// TIA Portal V20 export
FUNCTION_BLOCK "PartData"   // FB50063, LAD
// stored: MemoryReserve 100, Namespace Unit1.Em7, SetENOAutomatically false
   VAR
      statPulse { ExternalAccessible := 'False'; ExternalVisible := 'False'; ExternalWritable := 'False'} : Array[0..99] of Bool;
   END_VAR
   VAR_TEMP
      tempRetVal : Int;
   END_VAR
   VAR_TEMP   // added for the SCL form of the ladder/FBD networks
      _w1 : Bool;
      _w2 : Bool;
      _w3 : Bool;
      _w4 : Bool;
   END_VAR
BEGIN

REGION Network 1: Stack Table → Sepa Gripper
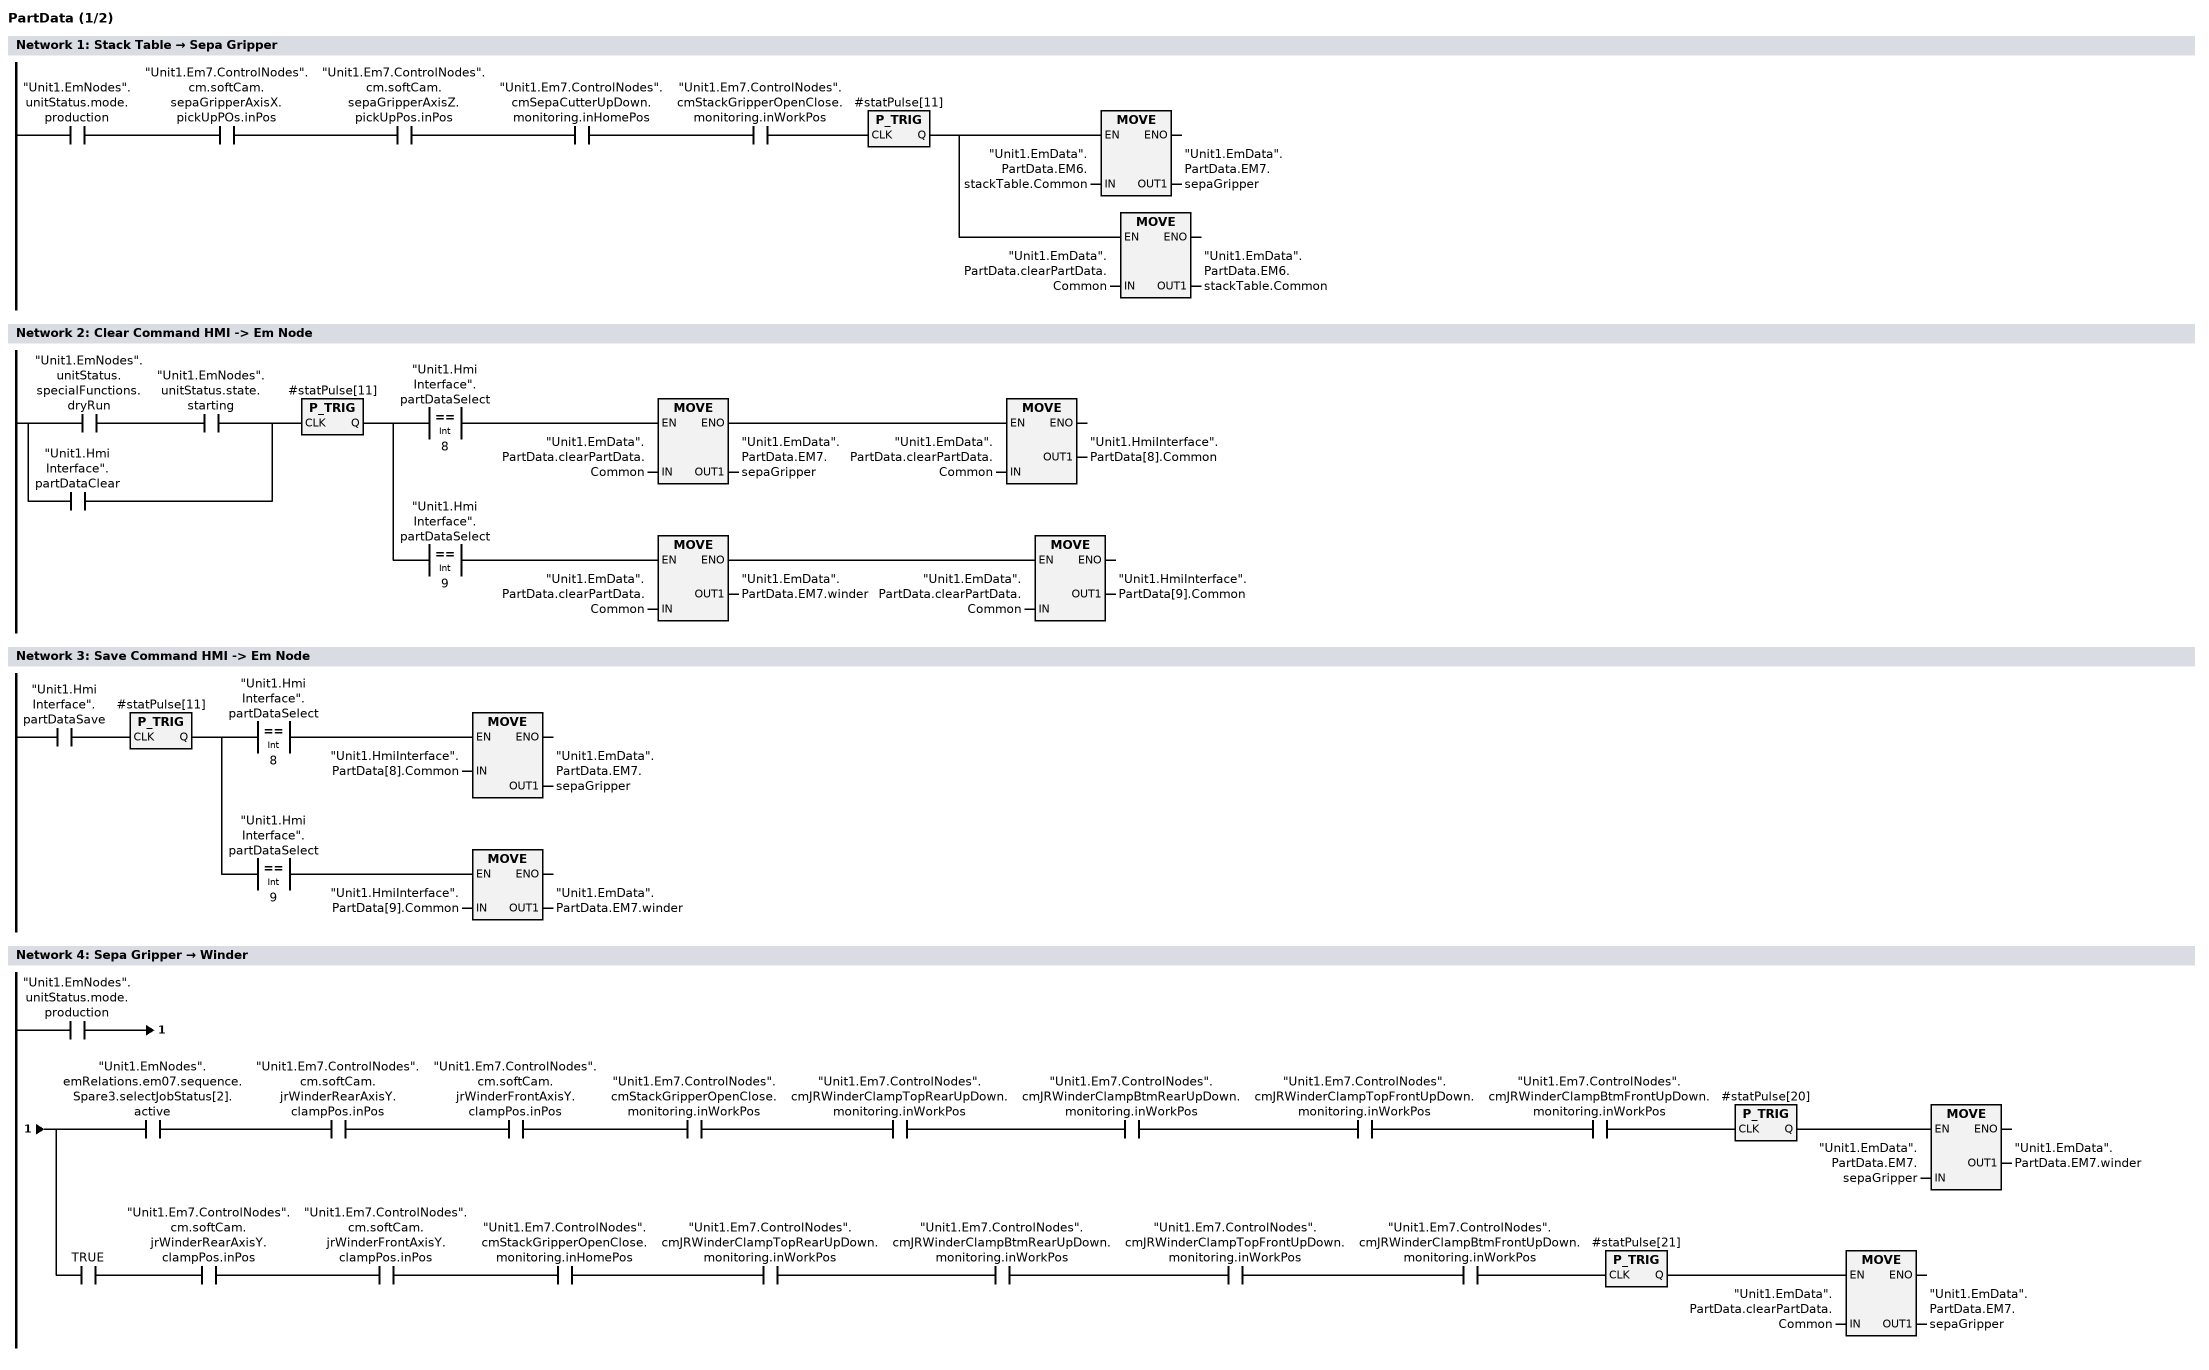
   RUNG wire#powerrail
      Contact( "Unit1.EmNodes".unitStatus.mode.production )
      Contact( "Unit1.Em7.ControlNodes".cm.softCam.sepaGripperAxisX.pickUpPOs.inPos )
      Contact( "Unit1.Em7.ControlNodes".cm.softCam.sepaGripperAxisZ.pickUpPos.inPos )
      Contact( "Unit1.Em7.ControlNodes".cmSepaCutterUpDown.monitoring.inHomePos )
      Contact( "Unit1.Em7.ControlNodes".cmStackGripperOpenClose.monitoring.inWorkPos )
      P_Trig( #statPulse[11] )
      wire#w1
      Move(in := "Unit1.EmData".PartData.EM6.stackTable.Common, out1 => "Unit1.EmData".PartData.EM7.sepaGripper)
   END_RUNG
   RUNG wire#w1
      Move(in := "Unit1.EmData".PartData.clearPartData.Common, out1 => "Unit1.EmData".PartData.EM6.stackTable.Common)
   END_RUNG
   // the same network as SCL:
   #_w1 := "Unit1.EmNodes".unitStatus.mode.production AND "Unit1.Em7.ControlNodes".cm.softCam.sepaGripperAxisX.pickUpPOs.inPos AND "Unit1.Em7.ControlNodes".cm.softCam.sepaGripperAxisZ.pickUpPos.inPos AND "Unit1.Em7.ControlNodes".cmSepaCutterUpDown.monitoring.inHomePos AND "Unit1.Em7.ControlNodes".cmStackGripperOpenClose.monitoring.inWorkPos;
   #_w2 := #_w1 AND NOT #statPulse[11];   // rising edge
   #statPulse[11] := #_w1;
   IF #_w2 THEN
       "Unit1.EmData".PartData.EM7.sepaGripper := "Unit1.EmData".PartData.EM6.stackTable.Common;
       "Unit1.EmData".PartData.EM6.stackTable.Common := "Unit1.EmData".PartData.clearPartData.Common;
   END_IF;
END_REGION

REGION Network 2: Clear Command HMI -> Em Node
   RUNG wire#powerrail
      Contact( "Unit1.EmNodes".unitStatus.specialFunctions.dryRun )
      Contact( "Unit1.EmNodes".unitStatus.state.starting )
      wire#w1
      P_Trig( #statPulse[11] )
      wire#w2
      { S7_Templates := "SrcType := Int" } EQ_Contact(in1 := "Unit1.HmiInterface".partDataSelect, in2 := 8)
      Move(in := "Unit1.EmData".PartData.clearPartData.Common, out1 => "Unit1.EmData".PartData.EM7.sepaGripper)
      Move(in := "Unit1.EmData".PartData.clearPartData.Common, out1 => "Unit1.HmiInterface".PartData[8].Common)
   END_RUNG
   RUNG wire#powerrail
      Contact( "Unit1.HmiInterface".partDataClear )
   END_RUNG wire#w1
   RUNG wire#w2
      { S7_Templates := "SrcType := Int" } EQ_Contact(in1 := "Unit1.HmiInterface".partDataSelect, in2 := 9)
      Move(in := "Unit1.EmData".PartData.clearPartData.Common, out1 => "Unit1.EmData".PartData.EM7.winder)
      Move(in := "Unit1.EmData".PartData.clearPartData.Common, out1 => "Unit1.HmiInterface".PartData[9].Common)
   END_RUNG
   // the same network as SCL:
   #_w1 := ("Unit1.EmNodes".unitStatus.specialFunctions.dryRun AND "Unit1.EmNodes".unitStatus.state.starting) OR "Unit1.HmiInterface".partDataClear;
   #_w2 := #_w1 AND NOT #statPulse[11];   // rising edge
   #statPulse[11] := #_w1;
   IF #_w2 AND ("Unit1.HmiInterface".partDataSelect = 8) THEN
       "Unit1.EmData".PartData.EM7.sepaGripper := "Unit1.EmData".PartData.clearPartData.Common;
       "Unit1.HmiInterface".PartData[8].Common := "Unit1.EmData".PartData.clearPartData.Common;
   END_IF;
   IF #_w2 AND ("Unit1.HmiInterface".partDataSelect = 9) THEN
       "Unit1.EmData".PartData.EM7.winder := "Unit1.EmData".PartData.clearPartData.Common;
       "Unit1.HmiInterface".PartData[9].Common := "Unit1.EmData".PartData.clearPartData.Common;
   END_IF;
END_REGION

REGION Network 3: Save Command HMI -> Em Node
   RUNG wire#powerrail
      Contact( "Unit1.HmiInterface".partDataSave )
      P_Trig( #statPulse[11] )
      wire#w1
      { S7_Templates := "SrcType := Int" } EQ_Contact(in1 := "Unit1.HmiInterface".partDataSelect, in2 := 8)
      Move(in := "Unit1.HmiInterface".PartData[8].Common, out1 => "Unit1.EmData".PartData.EM7.sepaGripper)
   END_RUNG
   RUNG wire#w1
      { S7_Templates := "SrcType := Int" } EQ_Contact(in1 := "Unit1.HmiInterface".partDataSelect, in2 := 9)
      Move(in := "Unit1.HmiInterface".PartData[9].Common, out1 => "Unit1.EmData".PartData.EM7.winder)
   END_RUNG
   // the same network as SCL:
   #_w1 := "Unit1.HmiInterface".partDataSave AND NOT #statPulse[11];   // rising edge
   #statPulse[11] := "Unit1.HmiInterface".partDataSave;
   IF #_w1 AND ("Unit1.HmiInterface".partDataSelect = 8) THEN
       "Unit1.EmData".PartData.EM7.sepaGripper := "Unit1.HmiInterface".PartData[8].Common;
   END_IF;
   IF #_w1 AND ("Unit1.HmiInterface".partDataSelect = 9) THEN
       "Unit1.EmData".PartData.EM7.winder := "Unit1.HmiInterface".PartData[9].Common;
   END_IF;
END_REGION

REGION Network 4: Sepa Gripper → Winder
   RUNG wire#powerrail
      Contact( "Unit1.EmNodes".unitStatus.mode.production )
      wire#w1
      Contact( "Unit1.EmNodes".emRelations.em07.sequence.Spare3.selectJobStatus[2].active )
      Contact( "Unit1.Em7.ControlNodes".cm.softCam.jrWinderRearAxisY.clampPos.inPos )
      Contact( "Unit1.Em7.ControlNodes".cm.softCam.jrWinderFrontAxisY.clampPos.inPos )
      Contact( "Unit1.Em7.ControlNodes".cmStackGripperOpenClose.monitoring.inWorkPos )
      Contact( "Unit1.Em7.ControlNodes".cmJRWinderClampTopRearUpDown.monitoring.inWorkPos )
      Contact( "Unit1.Em7.ControlNodes".cmJRWinderClampBtmRearUpDown.monitoring.inWorkPos )
      Contact( "Unit1.Em7.ControlNodes".cmJRWinderClampTopFrontUpDown.monitoring.inWorkPos )
      Contact( "Unit1.Em7.ControlNodes".cmJRWinderClampBtmFrontUpDown.monitoring.inWorkPos )
      P_Trig( #statPulse[20] )
      Move(in := "Unit1.EmData".PartData.EM7.sepaGripper, out1 => "Unit1.EmData".PartData.EM7.winder)
   END_RUNG
   RUNG wire#w1
      Contact( TRUE )
      Contact( "Unit1.Em7.ControlNodes".cm.softCam.jrWinderRearAxisY.clampPos.inPos )
      Contact( "Unit1.Em7.ControlNodes".cm.softCam.jrWinderFrontAxisY.clampPos.inPos )
      Contact( "Unit1.Em7.ControlNodes".cmStackGripperOpenClose.monitoring.inHomePos )
      Contact( "Unit1.Em7.ControlNodes".cmJRWinderClampTopRearUpDown.monitoring.inWorkPos )
      Contact( "Unit1.Em7.ControlNodes".cmJRWinderClampBtmRearUpDown.monitoring.inWorkPos )
      Contact( "Unit1.Em7.ControlNodes".cmJRWinderClampTopFrontUpDown.monitoring.inWorkPos )
      Contact( "Unit1.Em7.ControlNodes".cmJRWinderClampBtmFrontUpDown.monitoring.inWorkPos )
      P_Trig( #statPulse[21] )
      Move(in := "Unit1.EmData".PartData.clearPartData.Common, out1 => "Unit1.EmData".PartData.EM7.sepaGripper)
   END_RUNG
   // the same network as SCL:
   #_w1 := "Unit1.EmNodes".unitStatus.mode.production AND "Unit1.EmNodes".emRelations.em07.sequence.Spare3.selectJobStatus[2].active AND "Unit1.Em7.ControlNodes".cm.softCam.jrWinderRearAxisY.clampPos.inPos AND "Unit1.Em7.ControlNodes".cm.softCam.jrWinderFrontAxisY.clampPos.inPos AND "Unit1.Em7.ControlNodes".cmStackGripperOpenClose.monitoring.inWorkPos AND "Unit1.Em7.ControlNodes".cmJRWinderClampTopRearUpDown.monitoring.inWorkPos AND "Unit1.Em7.ControlNodes".cmJRWinderClampBtmRearUpDown.monitoring.inWorkPos AND "Unit1.Em7.ControlNodes".cmJRWinderClampTopFrontUpDown.monitoring.inWorkPos AND "Unit1.Em7.ControlNodes".cmJRWinderClampBtmFrontUpDown.monitoring.inWorkPos;
   #_w2 := #_w1 AND NOT #statPulse[20];   // rising edge
   #statPulse[20] := #_w1;
   IF #_w2 THEN "Unit1.EmData".PartData.EM7.winder := "Unit1.EmData".PartData.EM7.sepaGripper; END_IF;
   #_w3 := "Unit1.EmNodes".unitStatus.mode.production AND TRUE AND "Unit1.Em7.ControlNodes".cm.softCam.jrWinderRearAxisY.clampPos.inPos AND "Unit1.Em7.ControlNodes".cm.softCam.jrWinderFrontAxisY.clampPos.inPos AND "Unit1.Em7.ControlNodes".cmStackGripperOpenClose.monitoring.inHomePos AND "Unit1.Em7.ControlNodes".cmJRWinderClampTopRearUpDown.monitoring.inWorkPos AND "Unit1.Em7.ControlNodes".cmJRWinderClampBtmRearUpDown.monitoring.inWorkPos AND "Unit1.Em7.ControlNodes".cmJRWinderClampTopFrontUpDown.monitoring.inWorkPos AND "Unit1.Em7.ControlNodes".cmJRWinderClampBtmFrontUpDown.monitoring.inWorkPos;
   #_w4 := #_w3 AND NOT #statPulse[21];   // rising edge
   #statPulse[21] := #_w3;
   IF #_w4 THEN
       "Unit1.EmData".PartData.EM7.sepaGripper := "Unit1.EmData".PartData.clearPartData.Common;
   END_IF;
END_REGION

REGION Network 5: Winder → Sepa Gripper
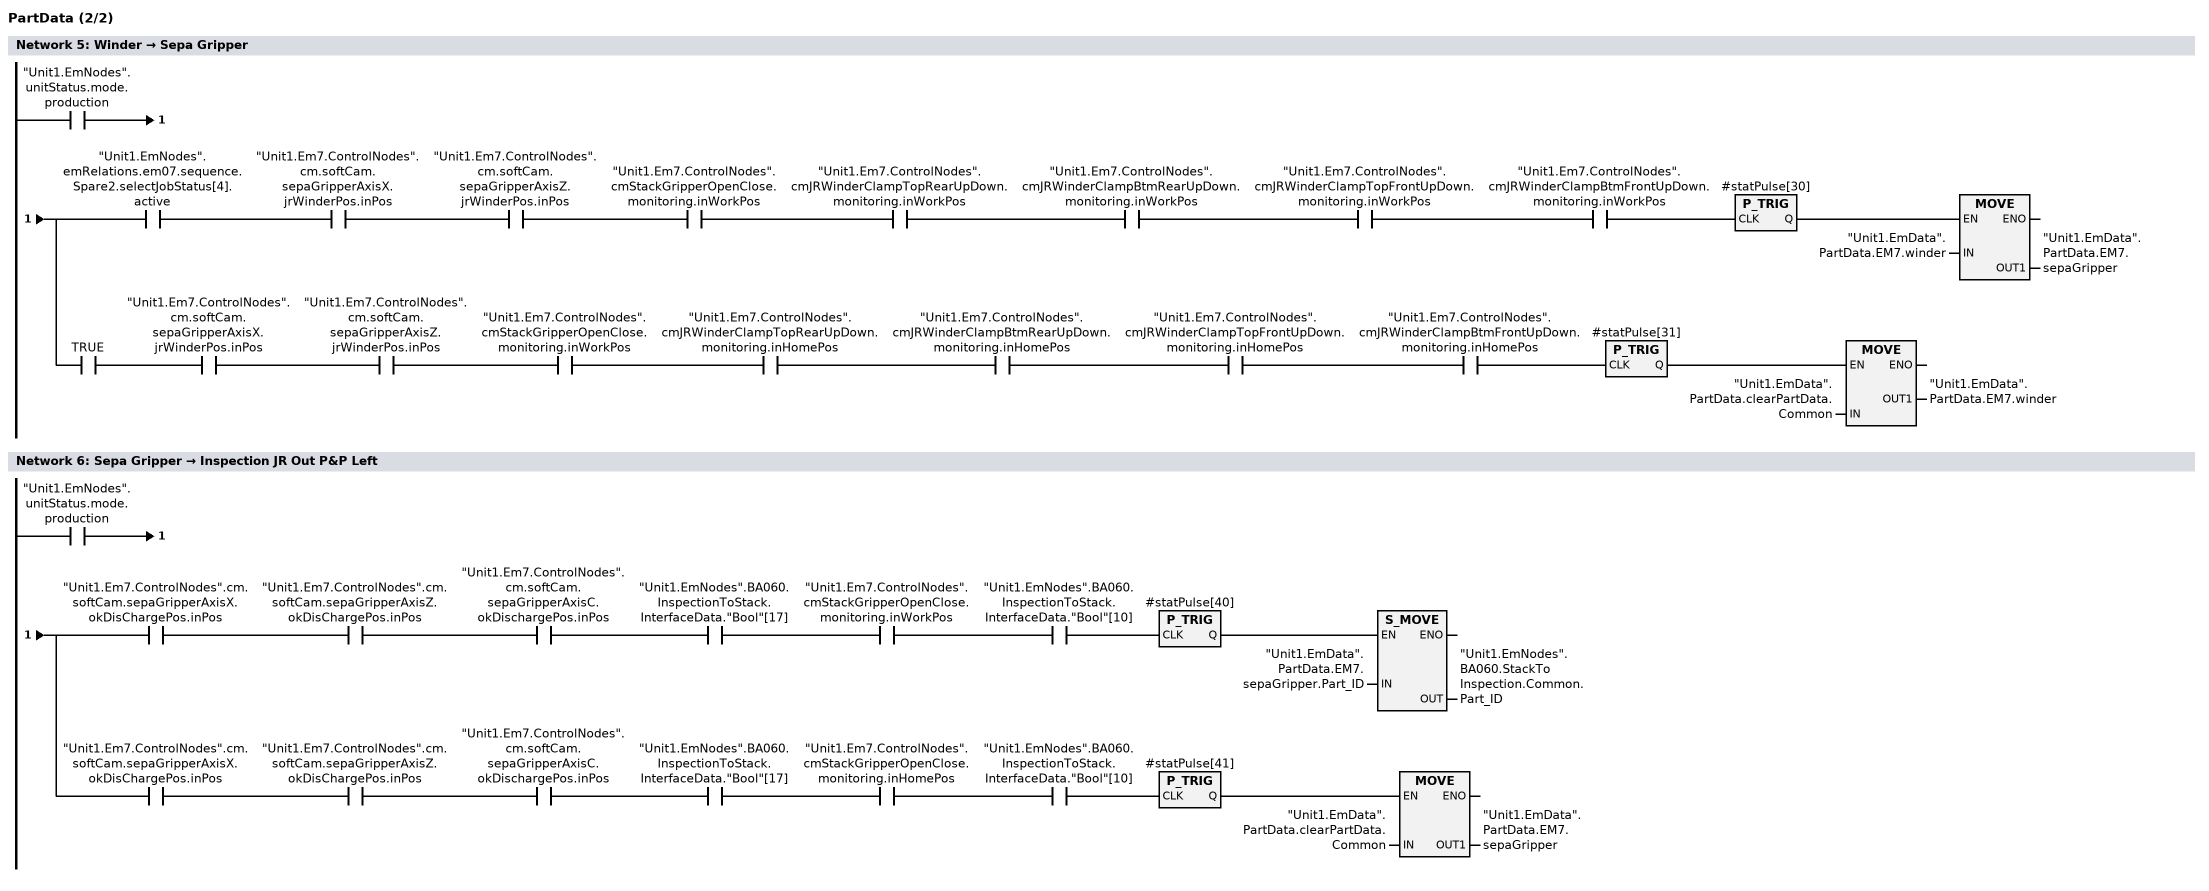
   RUNG wire#powerrail
      Contact( "Unit1.EmNodes".unitStatus.mode.production )
      wire#w1
      Contact( "Unit1.EmNodes".emRelations.em07.sequence.Spare2.selectJobStatus[4].active )
      Contact( "Unit1.Em7.ControlNodes".cm.softCam.sepaGripperAxisX.jrWinderPos.inPos )
      Contact( "Unit1.Em7.ControlNodes".cm.softCam.sepaGripperAxisZ.jrWinderPos.inPos )
      Contact( "Unit1.Em7.ControlNodes".cmStackGripperOpenClose.monitoring.inWorkPos )
      Contact( "Unit1.Em7.ControlNodes".cmJRWinderClampTopRearUpDown.monitoring.inWorkPos )
      Contact( "Unit1.Em7.ControlNodes".cmJRWinderClampBtmRearUpDown.monitoring.inWorkPos )
      Contact( "Unit1.Em7.ControlNodes".cmJRWinderClampTopFrontUpDown.monitoring.inWorkPos )
      Contact( "Unit1.Em7.ControlNodes".cmJRWinderClampBtmFrontUpDown.monitoring.inWorkPos )
      P_Trig( #statPulse[30] )
      Move(in := "Unit1.EmData".PartData.EM7.winder, out1 => "Unit1.EmData".PartData.EM7.sepaGripper)
   END_RUNG
   RUNG wire#w1
      Contact( TRUE )
      Contact( "Unit1.Em7.ControlNodes".cm.softCam.sepaGripperAxisX.jrWinderPos.inPos )
      Contact( "Unit1.Em7.ControlNodes".cm.softCam.sepaGripperAxisZ.jrWinderPos.inPos )
      Contact( "Unit1.Em7.ControlNodes".cmStackGripperOpenClose.monitoring.inWorkPos )
      Contact( "Unit1.Em7.ControlNodes".cmJRWinderClampTopRearUpDown.monitoring.inHomePos )
      Contact( "Unit1.Em7.ControlNodes".cmJRWinderClampBtmRearUpDown.monitoring.inHomePos )
      Contact( "Unit1.Em7.ControlNodes".cmJRWinderClampTopFrontUpDown.monitoring.inHomePos )
      Contact( "Unit1.Em7.ControlNodes".cmJRWinderClampBtmFrontUpDown.monitoring.inHomePos )
      P_Trig( #statPulse[31] )
      Move(in := "Unit1.EmData".PartData.clearPartData.Common, out1 => "Unit1.EmData".PartData.EM7.winder)
   END_RUNG
   // the same network as SCL:
   #_w1 := "Unit1.EmNodes".unitStatus.mode.production AND "Unit1.EmNodes".emRelations.em07.sequence.Spare2.selectJobStatus[4].active AND "Unit1.Em7.ControlNodes".cm.softCam.sepaGripperAxisX.jrWinderPos.inPos AND "Unit1.Em7.ControlNodes".cm.softCam.sepaGripperAxisZ.jrWinderPos.inPos AND "Unit1.Em7.ControlNodes".cmStackGripperOpenClose.monitoring.inWorkPos AND "Unit1.Em7.ControlNodes".cmJRWinderClampTopRearUpDown.monitoring.inWorkPos AND "Unit1.Em7.ControlNodes".cmJRWinderClampBtmRearUpDown.monitoring.inWorkPos AND "Unit1.Em7.ControlNodes".cmJRWinderClampTopFrontUpDown.monitoring.inWorkPos AND "Unit1.Em7.ControlNodes".cmJRWinderClampBtmFrontUpDown.monitoring.inWorkPos;
   #_w2 := #_w1 AND NOT #statPulse[30];   // rising edge
   #statPulse[30] := #_w1;
   IF #_w2 THEN "Unit1.EmData".PartData.EM7.sepaGripper := "Unit1.EmData".PartData.EM7.winder; END_IF;
   #_w3 := "Unit1.EmNodes".unitStatus.mode.production AND TRUE AND "Unit1.Em7.ControlNodes".cm.softCam.sepaGripperAxisX.jrWinderPos.inPos AND "Unit1.Em7.ControlNodes".cm.softCam.sepaGripperAxisZ.jrWinderPos.inPos AND "Unit1.Em7.ControlNodes".cmStackGripperOpenClose.monitoring.inWorkPos AND "Unit1.Em7.ControlNodes".cmJRWinderClampTopRearUpDown.monitoring.inHomePos AND "Unit1.Em7.ControlNodes".cmJRWinderClampBtmRearUpDown.monitoring.inHomePos AND "Unit1.Em7.ControlNodes".cmJRWinderClampTopFrontUpDown.monitoring.inHomePos AND "Unit1.Em7.ControlNodes".cmJRWinderClampBtmFrontUpDown.monitoring.inHomePos;
   #_w4 := #_w3 AND NOT #statPulse[31];   // rising edge
   #statPulse[31] := #_w3;
   IF #_w4 THEN "Unit1.EmData".PartData.EM7.winder := "Unit1.EmData".PartData.clearPartData.Common; END_IF;
END_REGION

REGION Network 6: Sepa Gripper → Inspection JR Out P&P Left
   RUNG wire#powerrail
      Contact( "Unit1.EmNodes".unitStatus.mode.production )
      wire#w1
      Contact( "Unit1.Em7.ControlNodes".cm.softCam.sepaGripperAxisX.okDisChargePos.inPos )
      Contact( "Unit1.Em7.ControlNodes".cm.softCam.sepaGripperAxisZ.okDisChargePos.inPos )
      Contact( "Unit1.Em7.ControlNodes".cm.softCam.sepaGripperAxisC.okDischargePos.inPos )
      Contact( "Unit1.EmNodes".BA060.InspectionToStack.InterfaceData."Bool"[17] )
      Contact( "Unit1.Em7.ControlNodes".cmStackGripperOpenClose.monitoring.inWorkPos )
      Contact( "Unit1.EmNodes".BA060.InspectionToStack.InterfaceData."Bool"[10] )
      P_Trig( #statPulse[40] )
      S_Move(in := "Unit1.EmData".PartData.EM7.sepaGripper.Part_ID, out => "Unit1.EmNodes".BA060.StackToInspection.Common.Part_ID)
   END_RUNG
   RUNG wire#w1
      Contact( "Unit1.Em7.ControlNodes".cm.softCam.sepaGripperAxisX.okDisChargePos.inPos )
      Contact( "Unit1.Em7.ControlNodes".cm.softCam.sepaGripperAxisZ.okDisChargePos.inPos )
      Contact( "Unit1.Em7.ControlNodes".cm.softCam.sepaGripperAxisC.okDischargePos.inPos )
      Contact( "Unit1.EmNodes".BA060.InspectionToStack.InterfaceData."Bool"[17] )
      Contact( "Unit1.Em7.ControlNodes".cmStackGripperOpenClose.monitoring.inHomePos )
      Contact( "Unit1.EmNodes".BA060.InspectionToStack.InterfaceData."Bool"[10] )
      P_Trig( #statPulse[41] )
      Move(in := "Unit1.EmData".PartData.clearPartData.Common, out1 => "Unit1.EmData".PartData.EM7.sepaGripper)
   END_RUNG
   // the same network as SCL:
   #_w1 := "Unit1.EmNodes".unitStatus.mode.production AND "Unit1.Em7.ControlNodes".cm.softCam.sepaGripperAxisX.okDisChargePos.inPos AND "Unit1.Em7.ControlNodes".cm.softCam.sepaGripperAxisZ.okDisChargePos.inPos AND "Unit1.Em7.ControlNodes".cm.softCam.sepaGripperAxisC.okDischargePos.inPos AND "Unit1.EmNodes".BA060.InspectionToStack.InterfaceData."Bool"[17] AND "Unit1.Em7.ControlNodes".cmStackGripperOpenClose.monitoring.inWorkPos AND "Unit1.EmNodes".BA060.InspectionToStack.InterfaceData."Bool"[10];
   #_w2 := #_w1 AND NOT #statPulse[40];   // rising edge
   #statPulse[40] := #_w1;
   IF #_w2 THEN
       "Unit1.EmNodes".BA060.StackToInspection.Common.Part_ID := "Unit1.EmData".PartData.EM7.sepaGripper.Part_ID;
   END_IF;
   #_w3 := "Unit1.EmNodes".unitStatus.mode.production AND "Unit1.Em7.ControlNodes".cm.softCam.sepaGripperAxisX.okDisChargePos.inPos AND "Unit1.Em7.ControlNodes".cm.softCam.sepaGripperAxisZ.okDisChargePos.inPos AND "Unit1.Em7.ControlNodes".cm.softCam.sepaGripperAxisC.okDischargePos.inPos AND "Unit1.EmNodes".BA060.InspectionToStack.InterfaceData."Bool"[17] AND "Unit1.Em7.ControlNodes".cmStackGripperOpenClose.monitoring.inHomePos AND "Unit1.EmNodes".BA060.InspectionToStack.InterfaceData."Bool"[10];
   #_w4 := #_w3 AND NOT #statPulse[41];   // rising edge
   #statPulse[41] := #_w3;
   IF #_w4 THEN
       "Unit1.EmData".PartData.EM7.sepaGripper := "Unit1.EmData".PartData.clearPartData.Common;
   END_IF;
END_REGION
END_FUNCTION_BLOCK
